# EPICS autosave request: apps/scalerApp/Db/scaler16m_addons_settings.req
# FILE... scaler16m_addons_settings.req
# USAGE.. transform Record fields autosave'd.

# needed to save OUTB-I
file transform_settings.req P=$(P)$(S)_cts1
file transform_settings.req P=$(P)$(S)_cts2
file transform_settings.req P=$(P)$(S)_norm1
file transform_settings.req P=$(P)$(S)_norm2

# FLNK from cts2 -> norm1
$(P)$(S)_cts2.FLNK
